TYPE ST_MCElementListWithParameter :
STRUCT
	arrNames 			: ARRAY  [1..GVL_BaseConstans.MAX_NUMBER_OF_ALL_ITEM] OF WSTRING;
	arrID				: ARRAY  [1..GVL_BaseConstans.MAX_NUMBER_OF_ALL_ITEM] OF UINT;
	iNumber				: INT;	//liczba elementów z parametrami
END_STRUCT
END_TYPE

(* stored: Version 1.1.0.1
   DUT ST_MCElementListWithParameter: Id {1029069d-be1c-0e74-0480-0f5bc5868154} *)
